PROGRAM Rezept_1
VAR
	// Abläufe
	Reaktor_1		:Grundablauf;
	Reaktor_2		:Grundablauf;
	Reaktor_3		:Grundablauf;
	Reaktor_4		:Grundablauf;
	Reaktor_5		:Grundablauf;
	Reaktor_6		:Grundablauf;
	Reaktor_7		:Grundablauf;
END_VAR

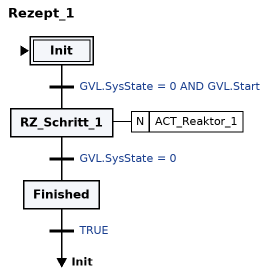
INITIAL_STEP Init:
END_STEP
TRANSITION FROM Init TO RZ_Schritt_1
    := GVL.SysState = 0 AND GVL.Start;
END_TRANSITION
STEP RZ_Schritt_1:
    ACT_Reaktor_1(N);
END_STEP
TRANSITION FROM RZ_Schritt_1 TO Finished
    := GVL.SysState = 0;
END_TRANSITION
STEP Finished:
END_STEP
TRANSITION FROM Finished TO Init
    := TRUE;
END_TRANSITION

ACTION ACT_Reaktor_1:
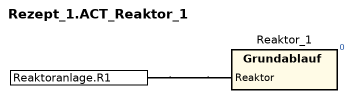
Reaktor_1(Reaktor := Reaktoranlage.R1); // Grundablauf
END_ACTION

ACTION ACT_Reaktor_2:
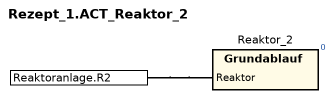
Reaktor_2(Reaktor := Reaktoranlage.R2); // Grundablauf
END_ACTION

ACTION ACT_Reaktor_3:
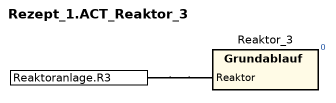
Reaktor_3(Reaktor := Reaktoranlage.R3); // Grundablauf
END_ACTION

ACTION ACT_Reaktor_4:
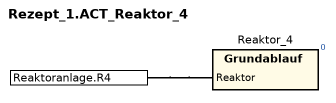
Reaktor_4(Reaktor := Reaktoranlage.R4); // Grundablauf
END_ACTION

ACTION ACT_Reaktor_5:
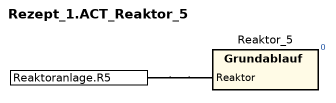
Reaktor_5(Reaktor := Reaktoranlage.R5); // Grundablauf
END_ACTION

ACTION ACT_Reaktor_6:
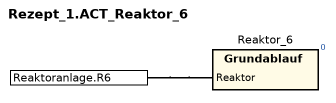
Reaktor_6(Reaktor := Reaktoranlage.R6); // Grundablauf
END_ACTION

ACTION ACT_Reaktor_7:
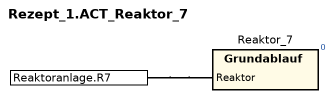
Reaktor_7(Reaktor := Reaktoranlage.R7); // Grundablauf
END_ACTION

END_PROGRAM

(* stored: Version 1.1.0.1, ProductVersion 3.1.4024.12
   POU Rezept_1: Id {f7eb72b6-2f07-4eb3-b931-f3427d1f70d5}, SpecialFunc None
   Action ACT_Reaktor_1: Id {a725f8db-5877-4260-a47f-b2887634ecd1}
   Action ACT_Reaktor_2: Id {767ee068-6834-4c4b-a594-3e2fa8658520}
   Action ACT_Reaktor_3: Id {471e8741-cb51-469a-a12d-8833622f2d81}
   Action ACT_Reaktor_4: Id {202d021c-4ac0-4e8c-ad39-9587c654dad0}
   Action ACT_Reaktor_5: Id {3d90a760-533d-41a4-83fb-7acbf1ca428e}
   Action ACT_Reaktor_6: Id {fc791d02-b608-446b-b583-72a60cfeb264}
   Action ACT_Reaktor_7: Id {c5a36271-c5bc-427e-8e4d-328282dc97d8} *)
